(* CODESYS project Hopper.xml

Project tree, tasks and I/O mapping:
  function block Hopper [LD]
*)

// Hopper
FUNCTION_BLOCK Hopper
VAR_INPUT
	Enable: 			BOOL;
	MaxSensor: 			BOOL; 				// Photoelectric sensor at minimum level.
	MinSensor: 			BOOL; 				// Photoelectric sensor at maximum level.
END_VAR
VAR_OUTPUT
	IceLevelOkay: 		BOOL;
	NeedIce: 			BOOL;
	Fault: 				BOOL;
END_VAR
VAR
	_IceAboveMaximum: 	BOOL; 				// Helper bit that's TRUE if ice is above maximum level.
	_IceAboveMinimum: 	BOOL; 				// Helper bit that's TRUE if ice is above minimum level.
	_SensorFault: 		BOOL;
END_VAR

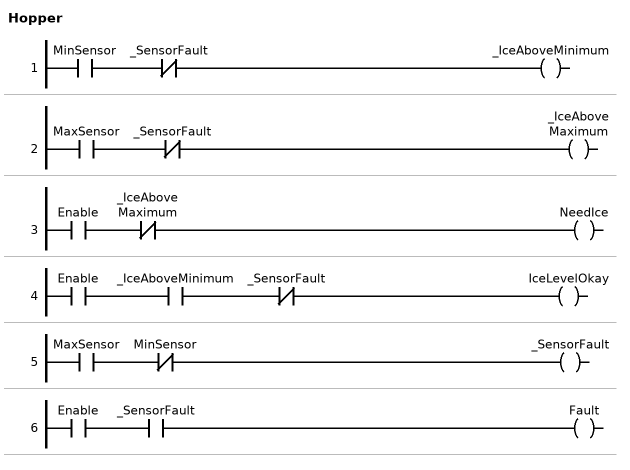
// NETWORK 1
_IceAboveMinimum := MinSensor AND NOT _SensorFault;

// NETWORK 2
_IceAboveMaximum := MaxSensor AND NOT _SensorFault;

// NETWORK 3
NeedIce := Enable AND NOT _IceAboveMaximum;

// NETWORK 4
IceLevelOkay := Enable AND _IceAboveMinimum AND NOT _SensorFault;

// NETWORK 5
_SensorFault := MaxSensor AND NOT MinSensor;

// NETWORK 6
Fault := Enable AND _SensorFault;

END_FUNCTION_BLOCK
